FUNCTION_BLOCK RunAxisAoiView EXTENDS RunAxisInspection
VAR
	
END_VAR

SUPER^();

CASE outputState OF
	eSpecialStates.SLAVE_ENTER_PROCEDURE:
		IF SlotBase^.Valid THEN
			bSerialTransition := TRUE;
		ELSE
			NextState := eSpecialStates.SLAVE_WORK_DONE;
		END_IF
	16#201:
		//align
		IF sideAligner^.Execute(argCommand:= eCylinderCommands.COMMAND_B) THEN
			NextState := eSpecialStates.SLAVE_AXIS_INSPECTION_ENTER;
		END_IF
	//----------------------------------
	eSpecialStates.SLAVE_AXIS_INSPECTION_EXIT:
		//release
		IF sideAligner^.Execute(eCylinderCommands.COMMAND_A) THEN
			NextState := eSpecialStates.SLAVE_WORK_DONE;
		END_IF
END_CASE

METHOD Initialize : BOOL
VAR_INPUT
END_VAR
//default initialization sequence
CASE outputState OF 
	eSpecialStates.INITIAL_BEGIN:
		NextState := eSpecialStates.INITIAL_STATE_7;
END_CASE

Initialize := SUPER^.Initialize();
END_METHOD

END_FUNCTION_BLOCK

(* stored: Version 1.1.0.1, ProductVersion 3.1.4022.10
   POU RunAxisAoiView: Id {dd3c82d7-e0e7-490b-93f3-e200f9619a5e}, SpecialFunc None
   Method Initialize: Id {bce0c290-06e8-4f8e-9747-fe861d1b9107} *)
